{attribute 'qualified_only'}
TYPE ePsbCtRange :
(
	_100A := 100,
	_250A := 250,
	_400A := 400,
	_630A := 630,
	_1000A := 1000,
	_1500A := 1500,
	_2000A := 2000,
	_4000A := 4000
) UINT := _1000A;
END_TYPE

(* stored: Version 1.1.0.1, ProductVersion 3.1.4024.12
   DUT ePsbCtRange: Id {dbd7b08d-cfe9-4265-8e86-e00a4eb97c56} *)
